// TIA Portal V20 export
TYPE "typeCmControlNode"
// stored: Namespace Unit1.Em9
   STRUCT
      interlock : "Unit1.Em9.typeCmControlNodeInterlock";
   END_STRUCT;
END_TYPE
